FUNCTION_BLOCK T_GripperModule EXTENDS FB_PackML_BaseModule IMPLEMENTS I_GripperModule
VAR
	_gripper : I_Gripper;
	_cylinder : I_Cylinder;
	
	cylinderComponent : T_CylinderComponent;
	
	productionMode : T_GripperProductionMode;
	maintenanceMode : T_GripperMaintenanceMode;
	manualMode : T_GripperManualMode;
END_VAR

METHOD GenericInitialise
VAR_INPUT
	Gripper : I_Gripper;
	Cylinder : I_Cylinder;
END_VAR
_gripper := Gripper;
_cylinder := Cylinder;
cylinderComponent.GenericInitialise(_cylinder);

ComponentsCollection.AddComponent(cylinderComponent);
END_METHOD

END_FUNCTION_BLOCK

(* stored: Version 1.1.0.1, ProductVersion 3.1.4024.12
   POU T_GripperModule: Id {42e42228-1cf4-406c-b140-481db51bee8e}, SpecialFunc None
   Method GenericInitialise: Id {4d9f01f6-a7ef-4e32-88ae-a6cca647633f} *)
